// TIA Portal project "Foerderband" (V14)

(* hardware
DEVICE "S7-1200-Station_1"  S7-1200 Station
   slot 0: "Baugruppenträger_0"  S7-1200 Rack  Rack  V1.0
   slot 1: "PLC_1"  CPU 1214C DC/DC/DC  6ES7 214-1AG40-0XB0  V4.2
   slot 3: "AQ 1x12BIT_1"  AQ1 signal board  6ES7 232-4HA30-0XB0  V1.0
*)

// ===== PLC "PLC_1"  CPU 1214C DC/DC/DC =====

VAR_GLOBAL   // PLC tag table "Standard-Variablentabelle"
   "System_Byte" AT %MB100 : Byte;
   "FirstScan" AT %M100.0 : Bool;
   "DiagStatusUpdate" AT %M100.1 : Bool;
   "AlwaysTRUE" AT %M100.2 : Bool;
   "AlwaysFALSE" AT %M100.3 : Bool;
   "Clock_Byte" AT %MB110 : Byte;
   "Clock_10Hz" AT %M110.0 : Bool;
   "Clock_5Hz" AT %M110.1 : Bool;
   "Clock_2.5Hz" AT %M110.2 : Bool;
   "Clock_2Hz" AT %M110.3 : Bool;
   "Clock_1.25Hz" AT %M110.4 : Bool;
   "Clock_1Hz" AT %M110.5 : Bool;
   "Clock_0.625Hz" AT %M110.6 : Bool;
   "Clock_0.5Hz" AT %M110.7 : Bool;
   "B1" AT %I10.0 : Bool;   // Lichtgitter - Strahl 1
   "B2" AT %I10.1 : Bool;   // Lichtgitter - Strahl 2
   "B3" AT %I10.2 : Bool;   // Lichtgitter - Strahl 3
   "B4" AT %I10.3 : Bool;   // Lichtgitter - Strahl 4
   "B5" AT %I10.4 : Bool;   // Lichtgitter - Strahl 5
   "B6" AT %I10.5 : Bool;   // Lichtgitter - Strahl 6
   "B7" AT %I10.6 : Bool;   // Lichtgitter - Strahl 7
   "B8" AT %I10.7 : Bool;   // Lichtgitter - Strahl 8
   "S1" AT %I11.0 : Bool;   // Taster Start
   "Q1" AT %Q10.0 : Bool;   // Antrieb Förderband
   "Q2" AT %Q10.1 : Bool;   // Auswerfer 1
   "Q3" AT %Q10.2 : Bool;   // Auswerfer 2
   "Q4" AT %Q10.3 : Bool;   // Emitter
   "S2" AT %I11.1 : Bool;   // Not-Halt
   "AlleAusgänge" AT %QW0 : Word;
END_VAR

FUNCTION "fc_Foerderband" : Void   // FC1, FBD
{ S7_Optimized_Access := 'TRUE' }
VERSION : 0.1
BEGIN

REGION Network 1: Auswerfer
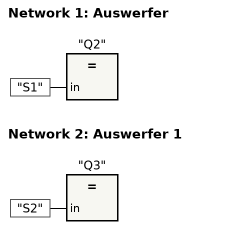
   "Q2" := "S1";
END_REGION

REGION Network 2: Auswerfer 1
   "Q3" := "S2";
END_REGION
END_FUNCTION

ORGANIZATION_BLOCK "Main"   // OB1, LAD, ProgramCycle
TITLE = "Main Program Sweep (Cycle)"
{ S7_Optimized_Access := 'TRUE' }
VERSION : 0.1
   VAR_INPUT
      Initial_Call : Bool;   // Initial call of this OB
      Remanence : Bool;   // =True, if remanent data are available
   END_VAR
BEGIN

REGION Network 1
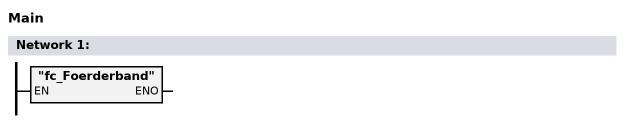
   RUNG wire#powerrail
      "fc_Foerderband"()
   END_RUNG
   // the same network as SCL:
   "fc_Foerderband"();
END_REGION
END_ORGANIZATION_BLOCK

ORGANIZATION_BLOCK "Startup"   // OB100, SCL, Startup
TITLE = "Complete Restart"
{ S7_Optimized_Access := 'TRUE' }
VERSION : 0.1
   VAR_INPUT
      LostRetentive : Bool;   // True if retentive data are lost
      LostRTC : Bool;   // True if date and time are lost
   END_VAR
BEGIN
   "AlleAusgänge" := 16#0000;
END_ORGANIZATION_BLOCK